Fanuc KAREL source: compact_preamble.KL

PROGRAM KA00066
%NOLOCKGROUP
VAR
SRC : XYZWPR;DST : XYZWPR
BEGIN
SRC.X=1.0
DST=SRC
END KA00066
